INTERFACE I_Extension EXTENDS I_Disposable, I_HostContent, I_HostInputPorts, I_HostOutputPorts, I_HostAlarms, I_HostParameters, I_HostMetadata, I_EventEmitter, I_Deserializable, I_Serializable

METHOD PUBLIC Accept
VAR_INPUT
	Visitor : I_ExtensionVisitor;
END_VAR
END_METHOD

PROPERTY PUBLIC Name : T_MAXSTRING
GET
END_GET
END_PROPERTY

END_INTERFACE

(* stored: Version 1.1.0.1, ProductVersion 3.1.4024.12
   Itf I_Extension: Id {3d8dc94f-e048-0570-13e2-c0ce07561e77}
   Method Accept: Id {280b39aa-7f93-0202-1dd6-de277e202a9e}
   Property Name: Id {810bedaa-c827-0105-38a9-63b394606d2a}
   Get Get: Id {45c513cd-293e-02ba-3f8b-9df680242548} *)
